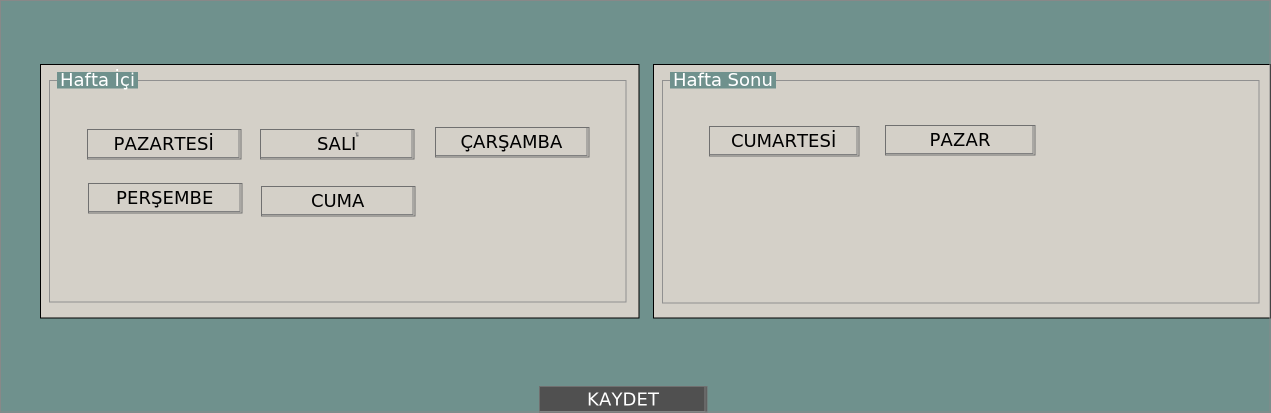
VISUALIZATION mesaigunleri_sayfa  // 1271x413
    Rectangle (653,64 618x254)
    Rectangle (40,64 599x254)
    GroupBox (49,72 577x230), "Hafta İçi"
        Button (38,57 154x30), "PAZARTESİ"
            toggle GVL_mesai_gun.pazartesi
        Button (211,57 154x30), "SALI"
            toggle GVL_mesai_gun.sali
        Button (386,55 154x30), "ÇARŞAMBA"
            toggle GVL_mesai_gun.carsamba
        Button (39,111 154x30), "PERŞEMBE"
            toggle GVL_mesai_gun.persembe
        Button (212,114 154x30), "CUMA"
            toggle GVL_mesai_gun.cuma
    GroupBox (662,72 597x231), "Hafta Sonu"
        Button (47,54 150x30), "CUMARTESİ"
            toggle GVL_mesai_gun.cumartesi
        Button (223,53 150x30), "PAZAR"
            toggle GVL_mesai_gun.pazar
    Button (539,386 168x27), "KAYDET"
        tap GVL_mesai_gun.kaydet
        OnMouseClick: change screen: MesaiSaat_sayfa
    Button (357,135 1x0)
END_VISUALIZATION

(* stored: Version 1.1.0.1, ProductVersion 3.1.4024.12
   Visu mesaigunleri_sayfa: Id {031f630b-033a-4e0e-9b0a-7d0d87491cbe} *)
